FUNCTION_BLOCK ABSTRACT FB_KNXnetIP_Device_Abstract
VAR_INPUT
	stInKnxGroupAddress		: ST_KNX_GroupAddress;
	ipInKnxTunneling		: I_KNXnetIP_Tunneling;
	ipInKnxInterpreter		: I_KNX_DPT_Interpreter;
	ipInKnxBuilder			: I_KNX_DPT_Builder;
END_VAR

END_FUNCTION_BLOCK

(* stored: Version 1.1.0.1
   POU FB_KNXnetIP_Device_Abstract: Id {4a1e7d36-21b7-422a-9a0b-9ddf9f19d91f}, SpecialFunc None *)
